// TIA Portal V18 export
FUNCTION "SS1_A3_8AI_IO_Update" : Void   // FC11030, LAD
{ S7_Optimized_Access := 'TRUE' }
VERSION : 0.1
// stored: AutoNumber false, IsIECCheckEnabled false, SetENOAutomatically false, UDAEnableTagReadback false
BEGIN

REGION Network 1: AI0
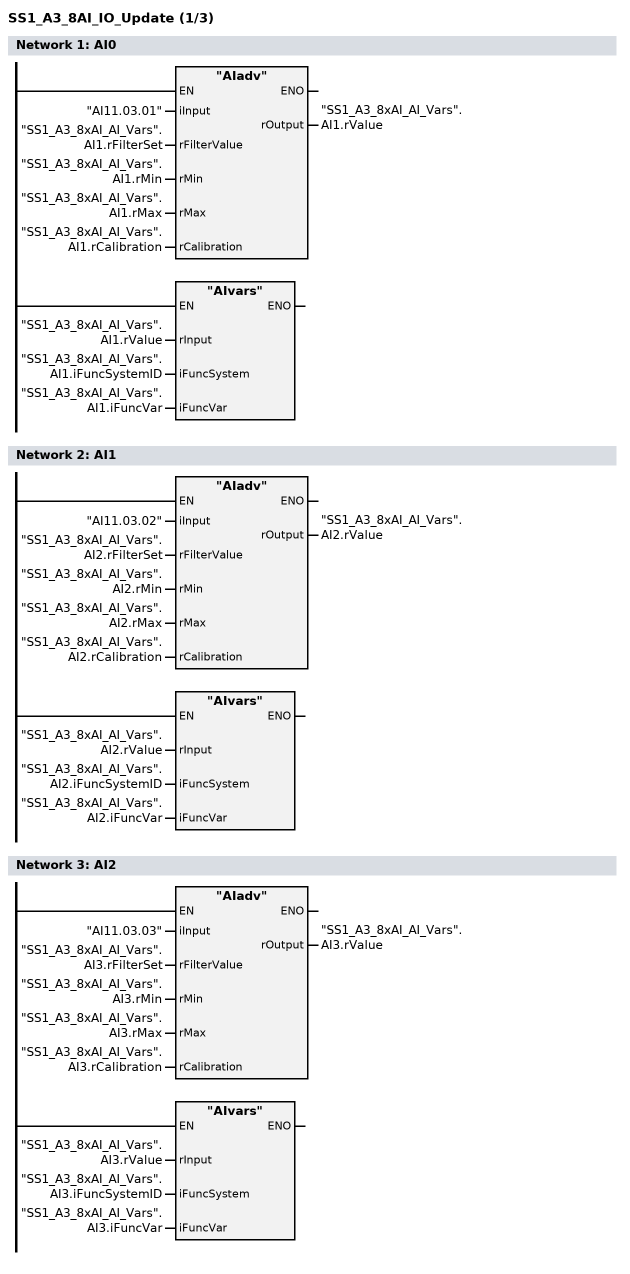
   RUNG wire#powerrail
      "AIadv"(iInput := "AI11.03.01", rFilterValue := "SS1_A3_8xAI_AI_Vars".AI1.rFilterSet, rMin := "SS1_A3_8xAI_AI_Vars".AI1.rMin, rMax := "SS1_A3_8xAI_AI_Vars".AI1.rMax, rCalibration := "SS1_A3_8xAI_AI_Vars".AI1.rCalibration, rOutput => "SS1_A3_8xAI_AI_Vars".AI1.rValue)
   END_RUNG
   RUNG wire#powerrail
      "AIvars"(rInput := "SS1_A3_8xAI_AI_Vars".AI1.rValue, iFuncSystem := "SS1_A3_8xAI_AI_Vars".AI1.iFuncSystemID, iFuncVar := "SS1_A3_8xAI_AI_Vars".AI1.iFuncVar)
   END_RUNG
   // the same network as SCL:
   "AIadv"(iInput := "AI11.03.01",
           rFilterValue := "SS1_A3_8xAI_AI_Vars".AI1.rFilterSet,
           rMin := "SS1_A3_8xAI_AI_Vars".AI1.rMin,
           rMax := "SS1_A3_8xAI_AI_Vars".AI1.rMax,
           rCalibration := "SS1_A3_8xAI_AI_Vars".AI1.rCalibration,
           rOutput => "SS1_A3_8xAI_AI_Vars".AI1.rValue);
   "AIvars"(rInput := "SS1_A3_8xAI_AI_Vars".AI1.rValue,
            iFuncSystem := "SS1_A3_8xAI_AI_Vars".AI1.iFuncSystemID,
            iFuncVar := "SS1_A3_8xAI_AI_Vars".AI1.iFuncVar);
END_REGION

REGION Network 2: AI1
   RUNG wire#powerrail
      "AIadv"(iInput := "AI11.03.02", rFilterValue := "SS1_A3_8xAI_AI_Vars".AI2.rFilterSet, rMin := "SS1_A3_8xAI_AI_Vars".AI2.rMin, rMax := "SS1_A3_8xAI_AI_Vars".AI2.rMax, rCalibration := "SS1_A3_8xAI_AI_Vars".AI2.rCalibration, rOutput => "SS1_A3_8xAI_AI_Vars".AI2.rValue)
   END_RUNG
   RUNG wire#powerrail
      "AIvars"(rInput := "SS1_A3_8xAI_AI_Vars".AI2.rValue, iFuncSystem := "SS1_A3_8xAI_AI_Vars".AI2.iFuncSystemID, iFuncVar := "SS1_A3_8xAI_AI_Vars".AI2.iFuncVar)
   END_RUNG
   // the same network as SCL:
   "AIadv"(iInput := "AI11.03.02",
           rFilterValue := "SS1_A3_8xAI_AI_Vars".AI2.rFilterSet,
           rMin := "SS1_A3_8xAI_AI_Vars".AI2.rMin,
           rMax := "SS1_A3_8xAI_AI_Vars".AI2.rMax,
           rCalibration := "SS1_A3_8xAI_AI_Vars".AI2.rCalibration,
           rOutput => "SS1_A3_8xAI_AI_Vars".AI2.rValue);
   "AIvars"(rInput := "SS1_A3_8xAI_AI_Vars".AI2.rValue,
            iFuncSystem := "SS1_A3_8xAI_AI_Vars".AI2.iFuncSystemID,
            iFuncVar := "SS1_A3_8xAI_AI_Vars".AI2.iFuncVar);
END_REGION

REGION Network 3: AI2
   RUNG wire#powerrail
      "AIadv"(iInput := "AI11.03.03", rFilterValue := "SS1_A3_8xAI_AI_Vars".AI3.rFilterSet, rMin := "SS1_A3_8xAI_AI_Vars".AI3.rMin, rMax := "SS1_A3_8xAI_AI_Vars".AI3.rMax, rCalibration := "SS1_A3_8xAI_AI_Vars".AI3.rCalibration, rOutput => "SS1_A3_8xAI_AI_Vars".AI3.rValue)
   END_RUNG
   RUNG wire#powerrail
      "AIvars"(rInput := "SS1_A3_8xAI_AI_Vars".AI3.rValue, iFuncSystem := "SS1_A3_8xAI_AI_Vars".AI3.iFuncSystemID, iFuncVar := "SS1_A3_8xAI_AI_Vars".AI3.iFuncVar)
   END_RUNG
   // the same network as SCL:
   "AIadv"(iInput := "AI11.03.03",
           rFilterValue := "SS1_A3_8xAI_AI_Vars".AI3.rFilterSet,
           rMin := "SS1_A3_8xAI_AI_Vars".AI3.rMin,
           rMax := "SS1_A3_8xAI_AI_Vars".AI3.rMax,
           rCalibration := "SS1_A3_8xAI_AI_Vars".AI3.rCalibration,
           rOutput => "SS1_A3_8xAI_AI_Vars".AI3.rValue);
   "AIvars"(rInput := "SS1_A3_8xAI_AI_Vars".AI3.rValue,
            iFuncSystem := "SS1_A3_8xAI_AI_Vars".AI3.iFuncSystemID,
            iFuncVar := "SS1_A3_8xAI_AI_Vars".AI3.iFuncVar);
END_REGION

REGION Network 4: AI3
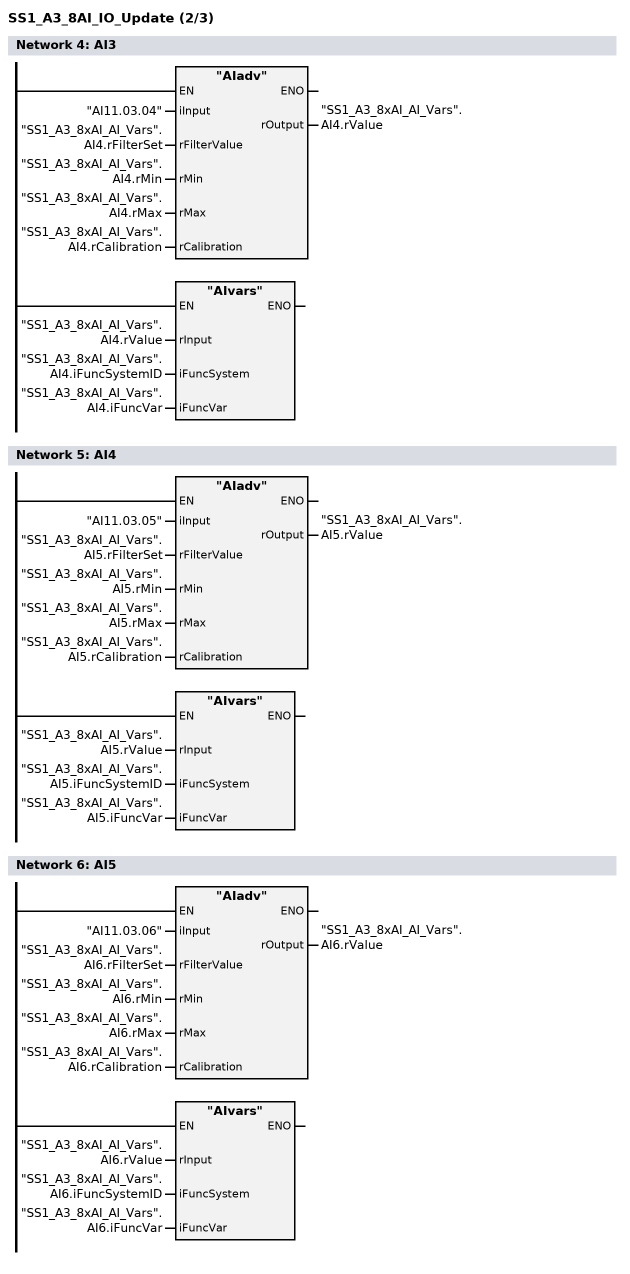
   RUNG wire#powerrail
      "AIadv"(iInput := "AI11.03.04", rFilterValue := "SS1_A3_8xAI_AI_Vars".AI4.rFilterSet, rMin := "SS1_A3_8xAI_AI_Vars".AI4.rMin, rMax := "SS1_A3_8xAI_AI_Vars".AI4.rMax, rCalibration := "SS1_A3_8xAI_AI_Vars".AI4.rCalibration, rOutput => "SS1_A3_8xAI_AI_Vars".AI4.rValue)
   END_RUNG
   RUNG wire#powerrail
      "AIvars"(rInput := "SS1_A3_8xAI_AI_Vars".AI4.rValue, iFuncSystem := "SS1_A3_8xAI_AI_Vars".AI4.iFuncSystemID, iFuncVar := "SS1_A3_8xAI_AI_Vars".AI4.iFuncVar)
   END_RUNG
   // the same network as SCL:
   "AIadv"(iInput := "AI11.03.04",
           rFilterValue := "SS1_A3_8xAI_AI_Vars".AI4.rFilterSet,
           rMin := "SS1_A3_8xAI_AI_Vars".AI4.rMin,
           rMax := "SS1_A3_8xAI_AI_Vars".AI4.rMax,
           rCalibration := "SS1_A3_8xAI_AI_Vars".AI4.rCalibration,
           rOutput => "SS1_A3_8xAI_AI_Vars".AI4.rValue);
   "AIvars"(rInput := "SS1_A3_8xAI_AI_Vars".AI4.rValue,
            iFuncSystem := "SS1_A3_8xAI_AI_Vars".AI4.iFuncSystemID,
            iFuncVar := "SS1_A3_8xAI_AI_Vars".AI4.iFuncVar);
END_REGION

REGION Network 5: AI4
   RUNG wire#powerrail
      "AIadv"(iInput := "AI11.03.05", rFilterValue := "SS1_A3_8xAI_AI_Vars".AI5.rFilterSet, rMin := "SS1_A3_8xAI_AI_Vars".AI5.rMin, rMax := "SS1_A3_8xAI_AI_Vars".AI5.rMax, rCalibration := "SS1_A3_8xAI_AI_Vars".AI5.rCalibration, rOutput => "SS1_A3_8xAI_AI_Vars".AI5.rValue)
   END_RUNG
   RUNG wire#powerrail
      "AIvars"(rInput := "SS1_A3_8xAI_AI_Vars".AI5.rValue, iFuncSystem := "SS1_A3_8xAI_AI_Vars".AI5.iFuncSystemID, iFuncVar := "SS1_A3_8xAI_AI_Vars".AI5.iFuncVar)
   END_RUNG
   // the same network as SCL:
   "AIadv"(iInput := "AI11.03.05",
           rFilterValue := "SS1_A3_8xAI_AI_Vars".AI5.rFilterSet,
           rMin := "SS1_A3_8xAI_AI_Vars".AI5.rMin,
           rMax := "SS1_A3_8xAI_AI_Vars".AI5.rMax,
           rCalibration := "SS1_A3_8xAI_AI_Vars".AI5.rCalibration,
           rOutput => "SS1_A3_8xAI_AI_Vars".AI5.rValue);
   "AIvars"(rInput := "SS1_A3_8xAI_AI_Vars".AI5.rValue,
            iFuncSystem := "SS1_A3_8xAI_AI_Vars".AI5.iFuncSystemID,
            iFuncVar := "SS1_A3_8xAI_AI_Vars".AI5.iFuncVar);
END_REGION

REGION Network 6: AI5
   RUNG wire#powerrail
      "AIadv"(iInput := "AI11.03.06", rFilterValue := "SS1_A3_8xAI_AI_Vars".AI6.rFilterSet, rMin := "SS1_A3_8xAI_AI_Vars".AI6.rMin, rMax := "SS1_A3_8xAI_AI_Vars".AI6.rMax, rCalibration := "SS1_A3_8xAI_AI_Vars".AI6.rCalibration, rOutput => "SS1_A3_8xAI_AI_Vars".AI6.rValue)
   END_RUNG
   RUNG wire#powerrail
      "AIvars"(rInput := "SS1_A3_8xAI_AI_Vars".AI6.rValue, iFuncSystem := "SS1_A3_8xAI_AI_Vars".AI6.iFuncSystemID, iFuncVar := "SS1_A3_8xAI_AI_Vars".AI6.iFuncVar)
   END_RUNG
   // the same network as SCL:
   "AIadv"(iInput := "AI11.03.06",
           rFilterValue := "SS1_A3_8xAI_AI_Vars".AI6.rFilterSet,
           rMin := "SS1_A3_8xAI_AI_Vars".AI6.rMin,
           rMax := "SS1_A3_8xAI_AI_Vars".AI6.rMax,
           rCalibration := "SS1_A3_8xAI_AI_Vars".AI6.rCalibration,
           rOutput => "SS1_A3_8xAI_AI_Vars".AI6.rValue);
   "AIvars"(rInput := "SS1_A3_8xAI_AI_Vars".AI6.rValue,
            iFuncSystem := "SS1_A3_8xAI_AI_Vars".AI6.iFuncSystemID,
            iFuncVar := "SS1_A3_8xAI_AI_Vars".AI6.iFuncVar);
END_REGION

REGION Network 7: AI6
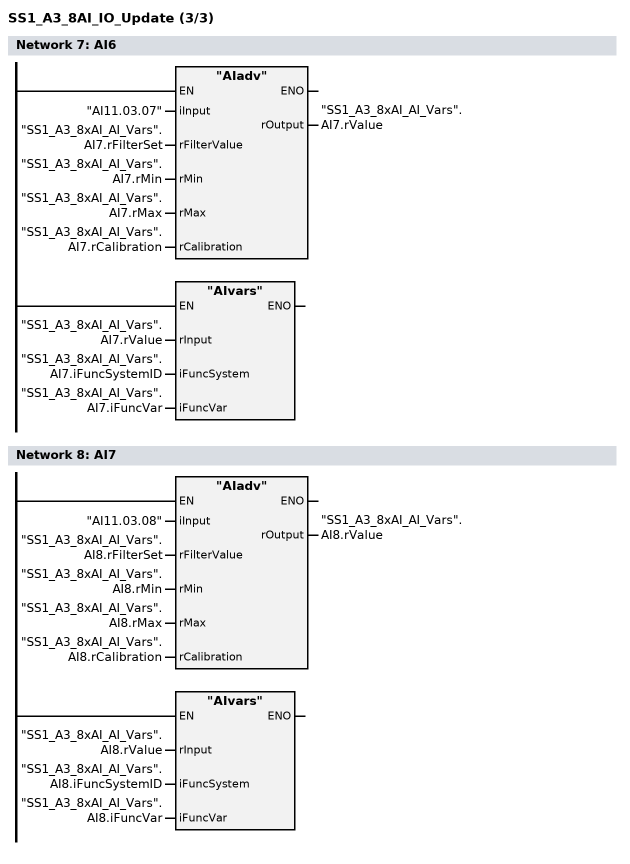
   RUNG wire#powerrail
      "AIadv"(iInput := "AI11.03.07", rFilterValue := "SS1_A3_8xAI_AI_Vars".AI7.rFilterSet, rMin := "SS1_A3_8xAI_AI_Vars".AI7.rMin, rMax := "SS1_A3_8xAI_AI_Vars".AI7.rMax, rCalibration := "SS1_A3_8xAI_AI_Vars".AI7.rCalibration, rOutput => "SS1_A3_8xAI_AI_Vars".AI7.rValue)
   END_RUNG
   RUNG wire#powerrail
      "AIvars"(rInput := "SS1_A3_8xAI_AI_Vars".AI7.rValue, iFuncSystem := "SS1_A3_8xAI_AI_Vars".AI7.iFuncSystemID, iFuncVar := "SS1_A3_8xAI_AI_Vars".AI7.iFuncVar)
   END_RUNG
   // the same network as SCL:
   "AIadv"(iInput := "AI11.03.07",
           rFilterValue := "SS1_A3_8xAI_AI_Vars".AI7.rFilterSet,
           rMin := "SS1_A3_8xAI_AI_Vars".AI7.rMin,
           rMax := "SS1_A3_8xAI_AI_Vars".AI7.rMax,
           rCalibration := "SS1_A3_8xAI_AI_Vars".AI7.rCalibration,
           rOutput => "SS1_A3_8xAI_AI_Vars".AI7.rValue);
   "AIvars"(rInput := "SS1_A3_8xAI_AI_Vars".AI7.rValue,
            iFuncSystem := "SS1_A3_8xAI_AI_Vars".AI7.iFuncSystemID,
            iFuncVar := "SS1_A3_8xAI_AI_Vars".AI7.iFuncVar);
END_REGION

REGION Network 8: AI7
   RUNG wire#powerrail
      "AIadv"(iInput := "AI11.03.08", rFilterValue := "SS1_A3_8xAI_AI_Vars".AI8.rFilterSet, rMin := "SS1_A3_8xAI_AI_Vars".AI8.rMin, rMax := "SS1_A3_8xAI_AI_Vars".AI8.rMax, rCalibration := "SS1_A3_8xAI_AI_Vars".AI8.rCalibration, rOutput => "SS1_A3_8xAI_AI_Vars".AI8.rValue)
   END_RUNG
   RUNG wire#powerrail
      "AIvars"(rInput := "SS1_A3_8xAI_AI_Vars".AI8.rValue, iFuncSystem := "SS1_A3_8xAI_AI_Vars".AI8.iFuncSystemID, iFuncVar := "SS1_A3_8xAI_AI_Vars".AI8.iFuncVar)
   END_RUNG
   // the same network as SCL:
   "AIadv"(iInput := "AI11.03.08",
           rFilterValue := "SS1_A3_8xAI_AI_Vars".AI8.rFilterSet,
           rMin := "SS1_A3_8xAI_AI_Vars".AI8.rMin,
           rMax := "SS1_A3_8xAI_AI_Vars".AI8.rMax,
           rCalibration := "SS1_A3_8xAI_AI_Vars".AI8.rCalibration,
           rOutput => "SS1_A3_8xAI_AI_Vars".AI8.rValue);
   "AIvars"(rInput := "SS1_A3_8xAI_AI_Vars".AI8.rValue,
            iFuncSystem := "SS1_A3_8xAI_AI_Vars".AI8.iFuncSystemID,
            iFuncVar := "SS1_A3_8xAI_AI_Vars".AI8.iFuncVar);
END_REGION
END_FUNCTION
